PROGRAM MAIN
VAR
END_VAR

(* 
	GOF 		Define an interface for creating an object, but let subclasses decide which class
				to instantiate. Factory Method lets a class defer instantiation to subclasses.
*)
P_FactoryPattern();

END_PROGRAM

(* stored: Version 1.1.0.1, ProductVersion 3.1.4024.12
   POU MAIN: Id {6e8820fe-31af-42d3-aaba-8e3a2c8f10cb}, SpecialFunc None *)
